FUNCTION_BLOCK FB_TestSuite3 EXTENDS FB_TestSuite
VAR_INPUT
END_VAR
VAR_OUTPUT
END_VAR
VAR
END_VAR

TestCase3A();

METHOD TestCase3A
VAR_INPUT
END_VAR
TEST('TestCase3A');

AssertTrue(TRUE, 'Condition is not true');
AssertTrue(TRUE, 'Condition is not true');

TEST_FINISHED();
END_METHOD

END_FUNCTION_BLOCK

(* stored: Version 1.1.0.1, ProductVersion 3.1.4024.12
   POU FB_TestSuite3: Id {4d879f8a-fdf2-40c8-8f49-cdcf59bed915}, SpecialFunc None
   Method TestCase3A: Id {ba8412ed-a485-4e34-a3cb-2c0117f9ef9e} *)
